// TwinCAT 3 PLC project Untitled1
// ProgramVersion: 3.1.4020.4
// libraries:
//   Tc2_Standard, * (Beckhoff Automation GmbH)
//   Tc2_System, * (Beckhoff Automation GmbH)
//   Tc2_Utilities, * (Beckhoff Automation GmbH)
//   Tc3_Module, * (Beckhoff Automation GmbH)
// project tree:
//   GVLs/ PersistentExample.TcGVL
//   / PlcTask.TcTTO
//   POUs/ CelsiusToFahrenheit.TcPOU, ForLoopExample.TcPOU, MAIN.TcPOU, MaintenanceCounter.TcPOU, SavePersistentVariables.TcPOU
// real-time tasks:
//   TASK PlcTask: cycle T#10ms, priority 20, ADS port 350

CONFIGURATION Untitled1
    RESOURCE PLC ON TwinCAT3
        TASK PlcTask(INTERVAL := T#10ms, PRIORITY := 20);
        PROGRAM MAIN WITH PlcTask : MAIN;
    END_RESOURCE
END_CONFIGURATION

// ---- GVLs/PersistentExample.TcGVL
{attribute 'qualified_only'}
VAR_GLOBAL PERSISTENT //to be persistent
	MyPersistentInteger : INT := 10;
END_VAR

VAR_GLOBAL // non persistent
	MyNonPersistentInteger : INT :=10;
END_VAR

// ---- POUs/MAIN.TcPOU
PROGRAM MAIN
VAR
END_VAR

//SavePersistentVariables();

END_PROGRAM

// ---- POUs/CelsiusToFahrenheit.TcPOU
FUNCTION CelsiusToFahrenheit  : REAL
VAR_INPUT
	TemperatureInCelsius :REAL;
END_VAR
VAR
	Temp:REAL;
END_VAR

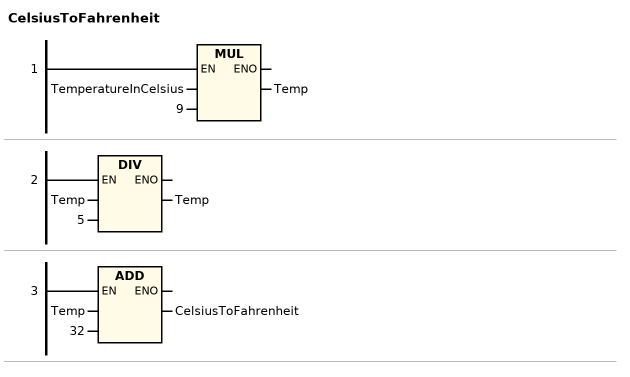
// NETWORK 1
Temp := TemperatureInCelsius * 9;

// NETWORK 2
Temp := Temp / 5;

// NETWORK 3
CelsiusToFahrenheit := Temp + 32;

END_FUNCTION

// ---- POUs/ForLoopExample.TcPOU
FUNCTION ForLoopExample : REAL
VAR_INPUT
END_VAR
VAR_IN_OUT
	MyArray : ARRAY [1..999] OF REAL;
END_VAR
VAR
	Sum:REAL;
	Index:INT;
END_VAR

Sum:=0;
FOR Index :=1 TO 999 BY 1 DO
	Sum := Sum + MyArray[Index];
END_FOR
ForLoopExample :=Sum / 999.0;

END_FUNCTION

// ---- POUs/MaintenanceCounter.TcPOU
FUNCTION_BLOCK MaintenanceCounter
VAR_INPUT
	 CU      : BOOL; (* Count Up *)
     RESET   : BOOL; (* Reset Counter to 0 *)
     PV      : DWORD; (* Counter Limit *)
END_VAR
VAR_OUTPUT
	Q       : BOOL; (* Counter reached the Limit *)
    CV      : DWORD; (* Current Counter Value *)
END_VAR
VAR PERSISTENT
	RisingEdge : R_TRIG;
	CurrentValue : DWORD;
END_VAR

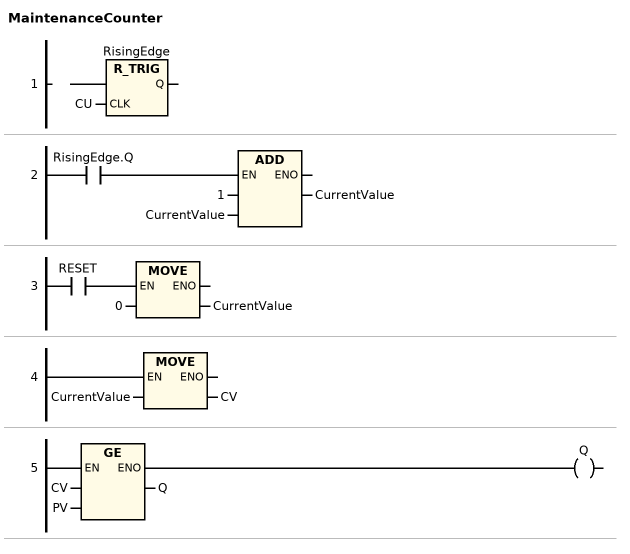
// NETWORK 1
RisingEdge(CLK := CU); // R_TRIG

// NETWORK 2
IF RisingEdge.Q THEN CurrentValue := 1 + CurrentValue; END_IF

// NETWORK 3
IF RESET THEN CurrentValue := 0; END_IF

// NETWORK 4
CV := CurrentValue;

// NETWORK 5
Q := CV >= PV;
Q := TRUE;

END_FUNCTION_BLOCK

// ---- POUs/SavePersistentVariables.TcPOU
PROGRAM SavePersistentVariables 
VAR
	WritePersistentDataFB : WritePersistentData;  //WritePersistentData FunctionBlock
	StartTON : TON;
	IntervalTON :TON;
END_VAR
VAR // added by the converter: edge detectors and wires of the graphical bodies
    _rt1 : R_TRIG;
END_VAR

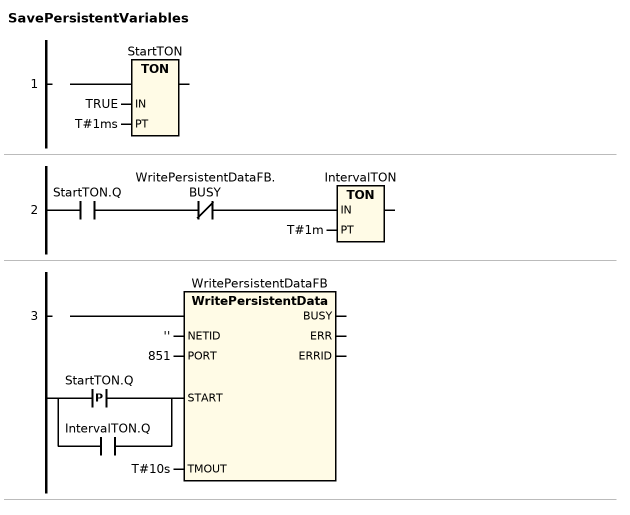
// NETWORK 1
StartTON(IN := TRUE, PT := T#1ms); // TON

// NETWORK 2
IntervalTON(IN := StartTON.Q AND NOT WritePersistentDataFB.BUSY, PT := T#1m); // TON

// NETWORK 3
_rt1(CLK := StartTON.Q);
WritePersistentDataFB(NETID := '', PORT := 851, START := _rt1.Q OR IntervalTON.Q, TMOUT := T#10s); // WritePersistentData

END_PROGRAM
